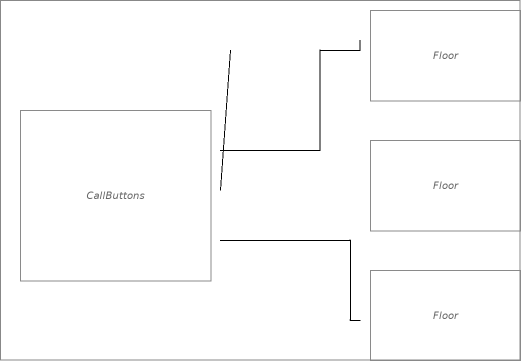
VISUALIZATION Visualization  // 521x361
    Frame (20,110 191x171)
        shows CallButtons(L1Call := MAIN.BT_FloorCall[1], L2Call := MAIN.BT_FloorCall[2], L3Call := MAIN.BT_FloorCall[3])
    Frame (370,10 151x91)
        shows Floor(LS_Floor := MAIN.LS_Floor[3])
        OnMouseClick: change screen: Screen3
    Frame (370,140 151x91)
        shows Floor(LS_Floor := MAIN.LS_Floor[2])
        OnMouseClick: change screen: Screen2
    Frame (370,270 151x91)
        shows Floor(LS_Floor := MAIN.LS_Floor[1])
        OnMouseClick: change screen: Screen1
    Polyline (220,150) (320,150) (320,50) (360,50) (360,40)
    Line (230,50) (220,190)
    Polyline (220,240) (350,240) (350,320) (360,320)
END_VISUALIZATION

(* stored: Version 1.1.0.1, ProductVersion 3.1.4024.11
   Visu Visualization: Id {950f217c-72e4-4728-89e4-6e96d124957e} *)
